INTERFACE INTERNAL I_ComponentNode EXTENDS I_Debug

PROPERTY _AsiComponent : I_Component
GET
END_GET
END_PROPERTY

PROPERTY INTERNAL _Entity : I_Entity
GET
END_GET
SET
END_SET
END_PROPERTY

PROPERTY INTERNAL _Next : I_ComponentNode
GET
END_GET
SET
END_SET
END_PROPERTY

PROPERTY INTERNAL _Prev : I_ComponentNode
GET
END_GET
SET
END_SET
END_PROPERTY

END_INTERFACE

(* stored: Version 1.1.0.1
   Itf I_ComponentNode: Id {293f8277-9be1-49c8-a36c-2a4c4768ebf2}
   Property _AsiComponent: Id {bee533d2-aa31-4bed-8f17-f26207ba6180}
   Get Get: Id {dee337c3-f9bf-42ee-9e16-82295ff3d5d5}
   Property _Entity: Id {670eeaaf-1eb0-40dc-8308-df4ae8a4caa3}
   Get Get: Id {03ff2e45-cbaa-495a-abce-74a0cb312780}
   Set Set: Id {118ba9f1-9041-4744-8ad9-0c110e8c3ce8}
   Property _Next: Id {fe269dd5-7715-4956-a298-8c9ea39c5bcb}
   Get Get: Id {eb0cb7a6-dbf9-4042-b35c-ff7f4f6b5171}
   Set Set: Id {817b0857-f5b8-49c5-96a8-c67347e8cc6e}
   Property _Prev: Id {b3c81385-4094-4de3-9289-9340b533a7d9}
   Get Get: Id {53c88c69-05c3-440e-a311-9d0ee9073f04}
   Set Set: Id {030fd2dd-439f-4b6a-b9ba-adba15c65969} *)
